// TwinCAT 3 PLC project Handler
// ProgramVersion: 3.1.4024.0
// libraries:
//   Tc2_Standard, * (Beckhoff Automation GmbH)
//   Tc2_System, * (Beckhoff Automation GmbH)
//   Tc2_Utilities, * (Beckhoff Automation GmbH)
//   Tc3_Module, * (Beckhoff Automation GmbH)
// project tree:
//   / GVL.TcGVL, PlcTask.TcTTO (not stored)
//   Library/Event/ E_Event.TcDUT, E_Type.TcDUT, FB_Event.TcPOU, I_Event.TcIO (not stored), ST_Event.TcDUT
//   Library/Handler/ FB_Handler.TcPOU, I_Handler.TcIO
//   POUs/ FB_Events.TcPOU, MAIN.TcPOU
// real-time tasks:
//   TASK PlcTask: cycle T#10ms, priority 20, ADS port 350

// ---- Library/Event/E_Event.TcDUT
{attribute 'qualified_only'}
{attribute 'strict'}
TYPE E_Event :
(
	Verbose		:= 0,
	Info		:= 1,
    Warning		:= 2,
    Error		:= 3,
    Critical	:= 4
)USINT;
END_TYPE

// ---- Library/Event/E_Type.TcDUT
{attribute 'qualified_only'}
{attribute 'strict'}
TYPE E_Type :
(
	None 			:= 0,
	Emergencey		:= 1,
	Error			:= 2,
	Stop			:= 3,
	Cycle			:= 4
)USINT;
END_TYPE

// ---- Library/Event/ST_Event.TcDUT
TYPE ST_Event :
STRUCT
	eType:		E_Type;
	eEvent:		E_Event;
	nTimestamp:	ULINT;
	nID:		DINT;
	sMessage:	STRING(255);
	sArguments:	STRING(255);
	sDefault:	STRING(255);
END_STRUCT
END_TYPE

// ---- GVL.TcGVL
VAR_GLOBAL
	Null:			PVOID:= 0;
END_VAR

// ---- Library/Handler/I_Handler.TcIO
INTERFACE I_Handler

METHOD PUBLIC M_Request
VAR_INPUT
	stEvent:			ST_Event;
END_VAR
END_METHOD

METHOD PUBLIC M_SetNext
VAR_INPUT
	iHandler:				I_Handler;
END_VAR
END_METHOD

END_INTERFACE

// ---- Library/Event/FB_Event.TcPOU
FUNCTION_BLOCK FB_Event IMPLEMENTS I_Event
VAR_INPUT
END_VAR
VAR_OUTPUT
END_VAR
VAR
	iHandler:			I_Handler;
	bVerbose:			BOOL;
	bInfo:				BOOL;
	bWarning:			BOOL;
	bError:				BOOL;
	bCritical:			BOOL;	
	stVerbose:			ST_Event;
	stInfo:				ST_Event;
	stWarning:			ST_Event;
	stError:			ST_Event;
	stCritical:			ST_Event;
END_VAR

IF bVerbose THEN
	bVerbose:= FALSE;
ELSE
	stVerbose.nTimestamp:= 0;
END_IF

IF bInfo THEN
	bInfo:= FALSE;	
ELSE
	stInfo.nTimestamp:= 0;		
END_IF

IF bWarning THEN
	bWarning:= FALSE;	
ELSE
	stWarning.nTimestamp:= 0;	
END_IF

IF bError THEN
	bError:= FALSE;	
ELSE
	stError.nTimestamp:= 0;	
END_IF
	
IF bCritical THEN
	bCritical:= FALSE;	
ELSE
	stCritical.nTimestamp:= 0;	
END_IF

METHOD M_Critical
VAR_INPUT
	eType:		E_Type;
	sMessage:	STRING(255);
	nID:		DINT;
END_VAR
bCritical:= TRUE;
IF stCritical.nTimestamp = 0 THEN
	stCritical.nTimestamp:= F_GetSystemTime();
END_IF
stCritical.eEvent:= E_Event.Critical;
stCritical.eType:= eType;
stCritical.sMessage:= sMessage;
stCritical.nID:= nID;

IF iHandler <> 0 THEN
	iHandler.M_Request(stCritical);
END_IF
END_METHOD

METHOD PUBLIC M_Error
VAR_INPUT
	eType:		E_Type;
	sMessage:	STRING(255);
	nID:		DINT;
END_VAR
bError:= TRUE;
IF stError.nTimestamp = 0 THEN
	stError.nTimestamp:= F_GetSystemTime();
END_IF
stError.eEvent:= E_Event.Critical;
stError.eType:= eType;
stError.sMessage:= sMessage;
stError.nID:= nID;

IF iHandler <> 0 THEN
	iHandler.M_Request(stError);
END_IF
END_METHOD

METHOD PUBLIC M_Info
VAR_INPUT
	eType:		E_Type;
	sMessage:	STRING(255);
	nID:		DINT;
END_VAR
bInfo:= TRUE;
IF stInfo.nTimestamp = 0 THEN
	stInfo.nTimestamp:= F_GetSystemTime();
END_IF
stInfo.eEvent:= E_Event.Critical;
stInfo.eType:= eType;
stInfo.sMessage:= sMessage;
stInfo.nID:= nID;

IF iHandler <> 0 THEN
	iHandler.M_Request(stInfo);
END_IF
END_METHOD

METHOD PUBLIC M_Verbose
VAR_INPUT
	eType:		E_Type;
	sMessage:	STRING(255);
	nID:		DINT;
END_VAR
bVerbose:= TRUE;
IF stVerbose.nTimestamp = 0 THEN
	stVerbose.nTimestamp:= F_GetSystemTime();
END_IF
stVerbose.eEvent:= E_Event.Critical;
stVerbose.eType:= eType;
stVerbose.sMessage:= sMessage;
stVerbose.nID:= nID;

IF iHandler <> 0 THEN
	iHandler.M_Request(stVerbose);
END_IF
END_METHOD

METHOD M_Warning
VAR_INPUT
	eType:		E_Type;
	sMessage:	STRING(255);
	nID:		DINT;
END_VAR
bWarning:= TRUE;
IF stWarning.nTimestamp = 0 THEN
	stWarning.nTimestamp:= F_GetSystemTime();
END_IF
stWarning.eEvent:= E_Event.Critical;
stWarning.eType:= eType;
stWarning.sMessage:= sMessage;
stWarning.nID:= nID;

IF iHandler <> 0 THEN
	iHandler.M_Request(stWarning);
END_IF
END_METHOD

PROPERTY PUBLIC P_Handler : I_Handler
GET
P_Handler:= iHandler;
END_GET
SET
iHandler:= P_Handler;
END_SET
END_PROPERTY

END_FUNCTION_BLOCK

// ---- Library/Handler/FB_Handler.TcPOU
FUNCTION_BLOCK ABSTRACT FB_Handler IMPLEMENTS I_Handler
VAR_INPUT
END_VAR
VAR_OUTPUT
END_VAR
VAR
	iNextHandler:			I_Handler;
END_VAR

//	The FB_Handler is an abstract function block that implements the I_Handler interface. 
//	It represents a handler in the Chain of Responsibility pattern,
//	where a request can be passed along a chain of potential handlers until one of them handles the request.
//	Each handler in the chain has the ability to either handle the request or pass it to the next handle

METHOD PUBLIC M_Request
VAR_INPUT
	stEvent:			ST_Event;		// event to be handled. 
END_VAR
// The M_Request method is used to handle the request.

IF iNextHandler <> 0 THEN
	// the request is passed to the next handler 
	iNextHandler.M_Request(stEvent);
END_IF
END_METHOD

METHOD PUBLIC M_SetNext
VAR_INPUT
	iHandler:				I_Handler;
END_VAR
// next handler in the chain
iNextHandler:= iHandler;
END_METHOD

END_FUNCTION_BLOCK

// ---- POUs/FB_Events.TcPOU
FUNCTION_BLOCK FB_Events EXTENDS FB_Handler
VAR_INPUT
END_VAR
VAR_OUTPUT
END_VAR
VAR
	nEvents:		INT;
	aEvents:		ARRAY [0..100] OF ST_Event;
END_VAR

SUPER^();

METHOD PRIVATE M_Find : INT
VAR_INPUT
	stEvent:			ST_Event;		// event to find
END_VAR
VAR
	nIndex: INT;
END_VAR
FOR nIndex:= 0 TO nEvents DO
	IF memcmp(ADR(aEvents[nEvents]), ADR(stEvent), SIZEOF(stEvent)) = 0 THEN
		M_Find:= nIndex;
		RETURN;
	END_IF
END_FOR
END_METHOD

METHOD PUBLIC M_Request
VAR_INPUT
	stEvent:			ST_Event;		// event to be handled. 
END_VAR
SUPER^.M_Request(stEvent);

IF nEvents < 100 THEN
	IF M_Find(stEvent) = 0 THEN
		aEvents[nEvents]:= stEvent;
		nEvents:= nEvents + 1;
	END_IF
END_IF
END_METHOD

END_FUNCTION_BLOCK

// ---- POUs/MAIN.TcPOU
PROGRAM MAIN
VAR
	fbEvent:		FB_Event;
	fbHandler:		FB_Events;
	bInit:			BOOL:= TRUE;;
	bEvent: 		BOOL;
END_VAR

IF bInit THEN
	bInit:= FALSE;
	fbEvent.P_Handler:= fbHandler;
END_IF

fbHandler();

IF bEvent THEN
	fbEvent.M_Critical(E_Type.Error, 'Message', 1);
END_IF

END_PROGRAM
